{attribute addProperty BoxType "EL3751-0000-0020"}
{attribute addProperty Id "SamplesAT %I*ARRAY [0..0] OF DINT324"}
{attribute addProperty CRC "1340537356"}
{attribute addProperty SizeInBites "32"}
{attribute addProperty SizeInBytes "4"}
TYPE PAI_Samples_4FE6FA0C :
STRUCT
	{attribute addProperty Name "Samples"}
	Samples AT %I* : ARRAY [0..0] OF DINT;
END_STRUCT
END_TYPE

(* stored: Version 1.2.0.0, ProductVersion 3.1.4024.9
   DUT PAI_Samples_4FE6FA0C: Id {2e0c6be1-0762-4d39-bd11-af4e06049492} *)
